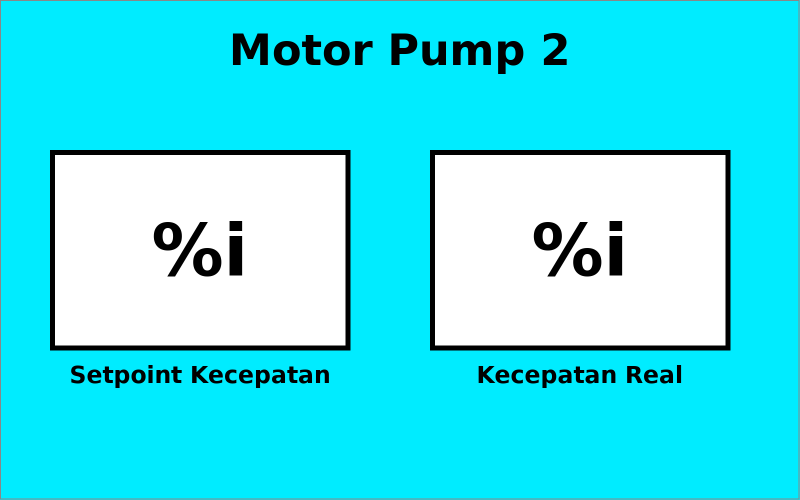
VISUALIZATION Screen_2_Sub_4  // 800x500
    Rectangle (0,0 800x500)
    Label (0,0 800x100), "Motor Pump 2"
    Rectangle (50,150 300x200), "%i", text variable: GVL.HMI_Motor_Pump_2_Input
        OnMouseClick: write GVL.HMI_Motor_Pump_2_Input via VisuDialogs.Numpad
    Label (50,350 300x50), "Setpoint Kecepatan"
    Label (430,350 300x50), "Kecepatan Real"
    Rectangle (430,150 300x200), "%i", text variable: GVL.HMI_Motor_Pump_2_Real
END_VISUALIZATION

(* stored: Version 1.1.0.1, ProductVersion 3.1.4024.12
   Visu Screen_2_Sub_4: Id {11ff093c-6a56-4d66-b81b-ae09ab1f46b1} *)
